# EPICS autosave request: softGlueApp/Db/ScalToStream_settings.req
$(P)$(H)scalToStream-$(N)_desc
$(P)$(H)scalToStream-$(N)_CHADV_Signal
$(P)$(H)scalToStream-$(N)_ADVDONE_Signal
$(P)$(H)scalToStream-$(N)_FULL_Signal
$(P)$(H)scalToStream-$(N)_RESET_Signal
$(P)$(H)scalToStream-$(N)_DMAWORDS
